// SIMATIC S7-200 project (STEP 7-Micro/WIN), CPU 224 AM REL 21.02

ORGANIZATION_BLOCK 主程序:OB1
TITLE=本MODBUS TCP 服务器库  可以建立两个 MODBUS TCP 服务器
// Socket：       填写1或者2通道（1=端口号502，2等于端口号503）
// MaxIO：        I 和Q 位最大数目（默认值128）
// MaxAI：        输入寄存器最大数目
// MaxHold：    保持寄存器最大数目
// ptrHold：       保持寄存器在V内存中的起始地址
// slaveAddr：  本服务端站号
// Error：           错误代码 =1 表示非法的数据地址 ， =2 表示错误的通信口 
// 
// 程序下载到PLC里面后需要重新上电
BEGIN
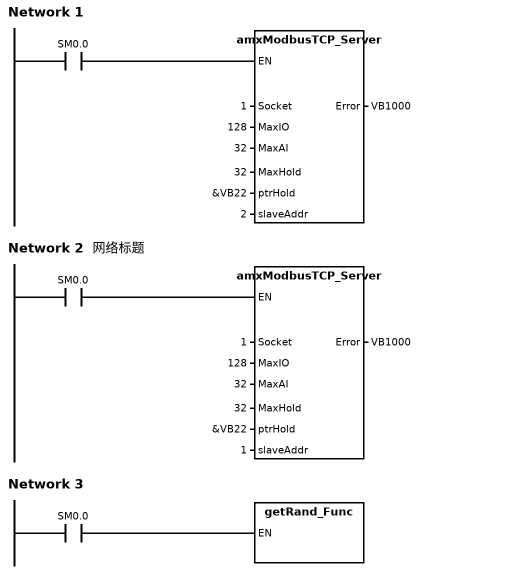
Network 1
LD     SM0.0
CALL   amxModbusTCP_Server:SBR1, 1, 128, 32, 32, &VB22, 2, VB1000
Network 2 // 网络标题
LD     SM0.0
CALL   amxModbusTCP_Server:SBR1, 1, 128, 32, 32, &VB22, 1, VB1000
Network 3
LD     SM0.0
CALL   getRand_Func:SBR0
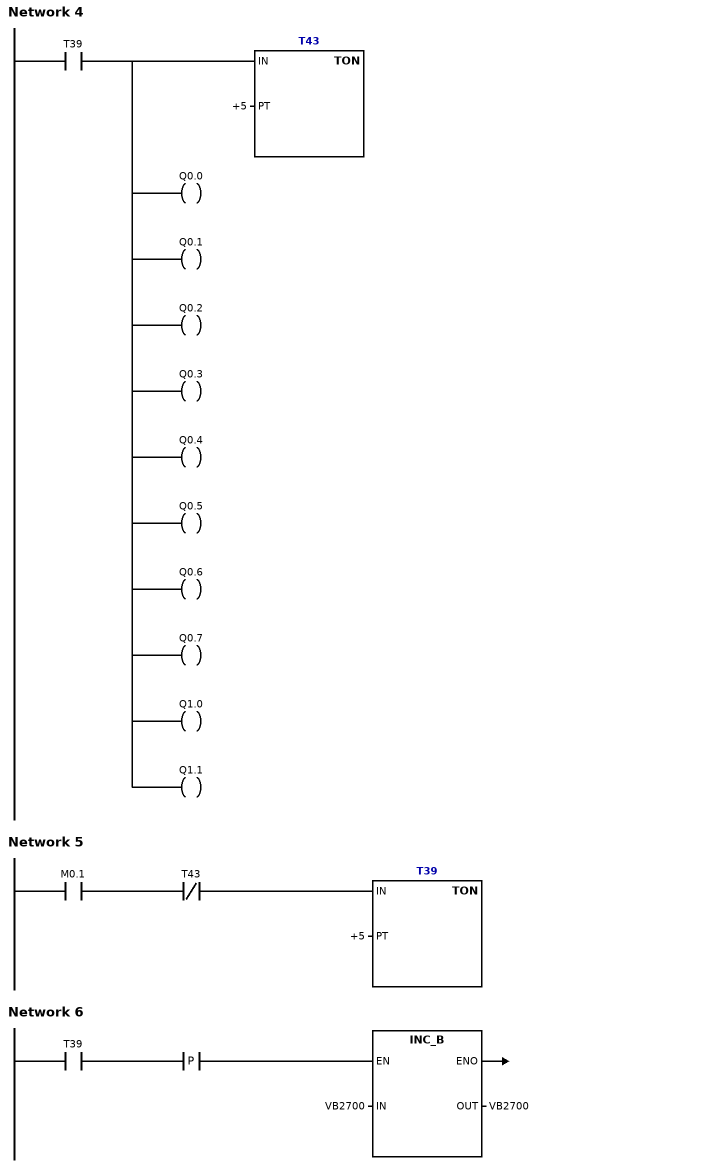
Network 4
LD     T39
TON    T43, +5
=      Q0.0
=      Q0.1
=      Q0.2
=      Q0.3
=      Q0.4
=      Q0.5
=      Q0.6
=      Q0.7
=      Q1.0
=      Q1.1
Network 5
LD     M0.1
AN     T43
TON    T39, +5
Network 6
LD     T39
EU
INCB   VB2700
END_ORGANIZATION_BLOCK

SUBROUTINE_BLOCK getRand_Func:SBR0
TITLE=
BEGIN
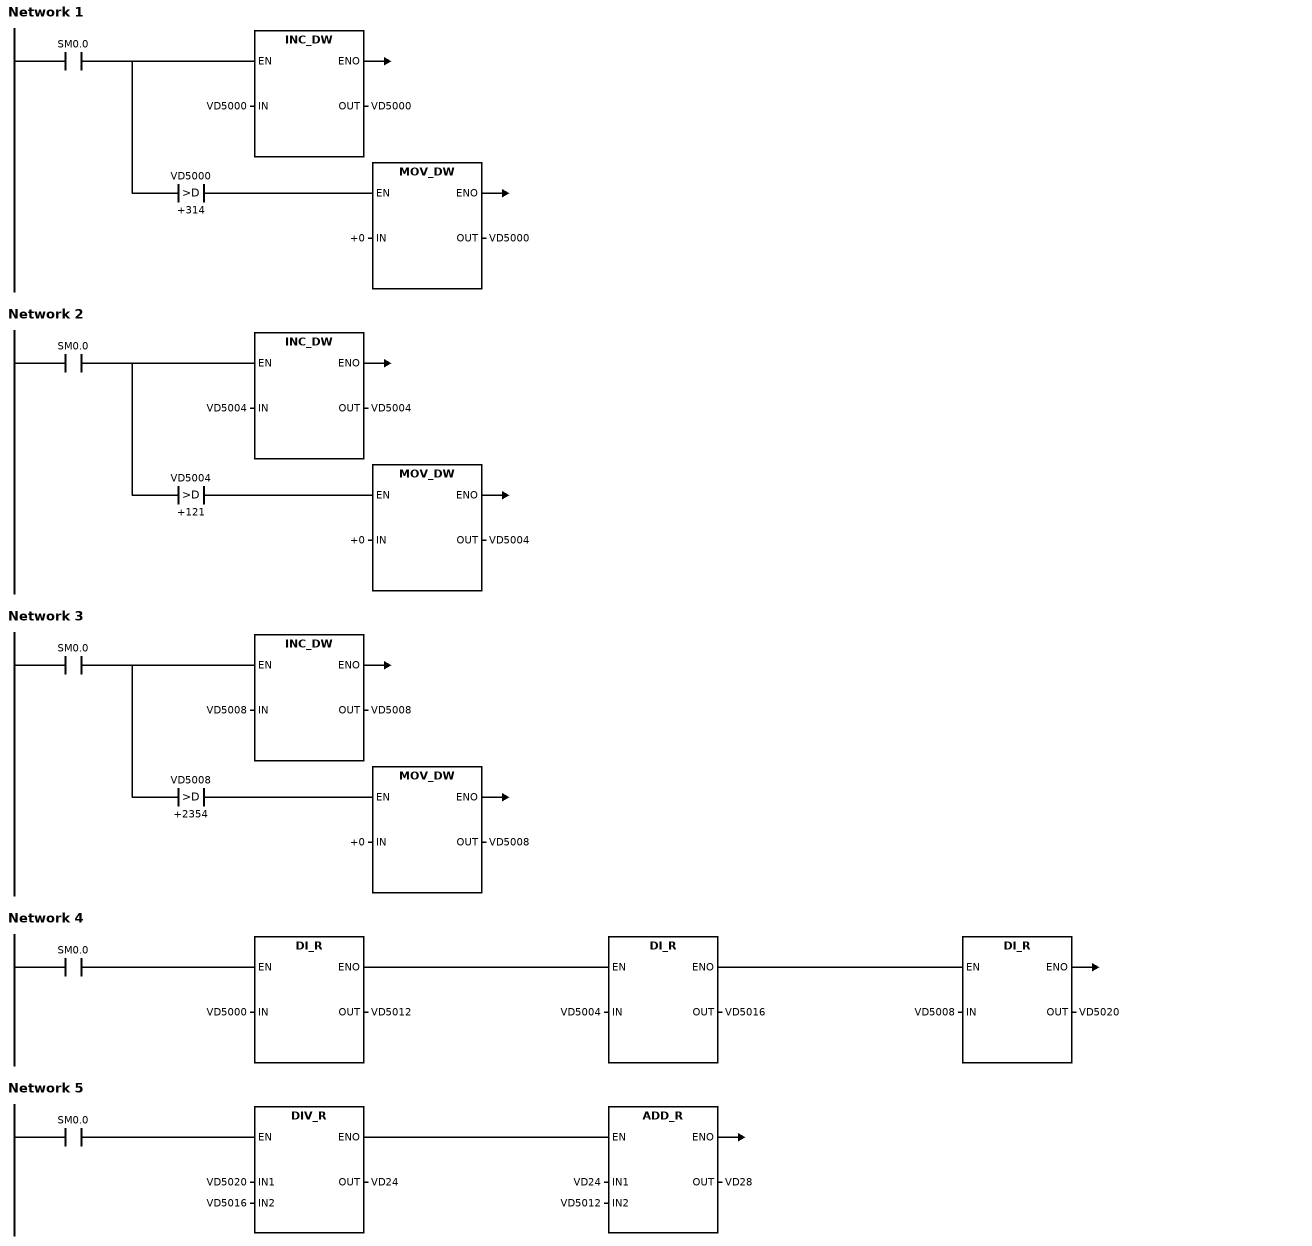
Network 1
LD     SM0.0
INCD   VD5000
AD>    VD5000, +314
MOVD   +0, VD5000
Network 2
LD     SM0.0
INCD   VD5004
AD>    VD5004, +121
MOVD   +0, VD5004
Network 3
LD     SM0.0
INCD   VD5008
AD>    VD5008, +2354
MOVD   +0, VD5008
Network 4
LD     SM0.0
DTR    VD5000, VD5012
AENO
DTR    VD5004, VD5016
AENO
DTR    VD5008, VD5020
Network 5
LD     SM0.0
MOVR   VD5020, VD24
AENO
/R     VD5016, VD24
AENO
MOVR   VD24, VD28
+R     VD5012, VD28
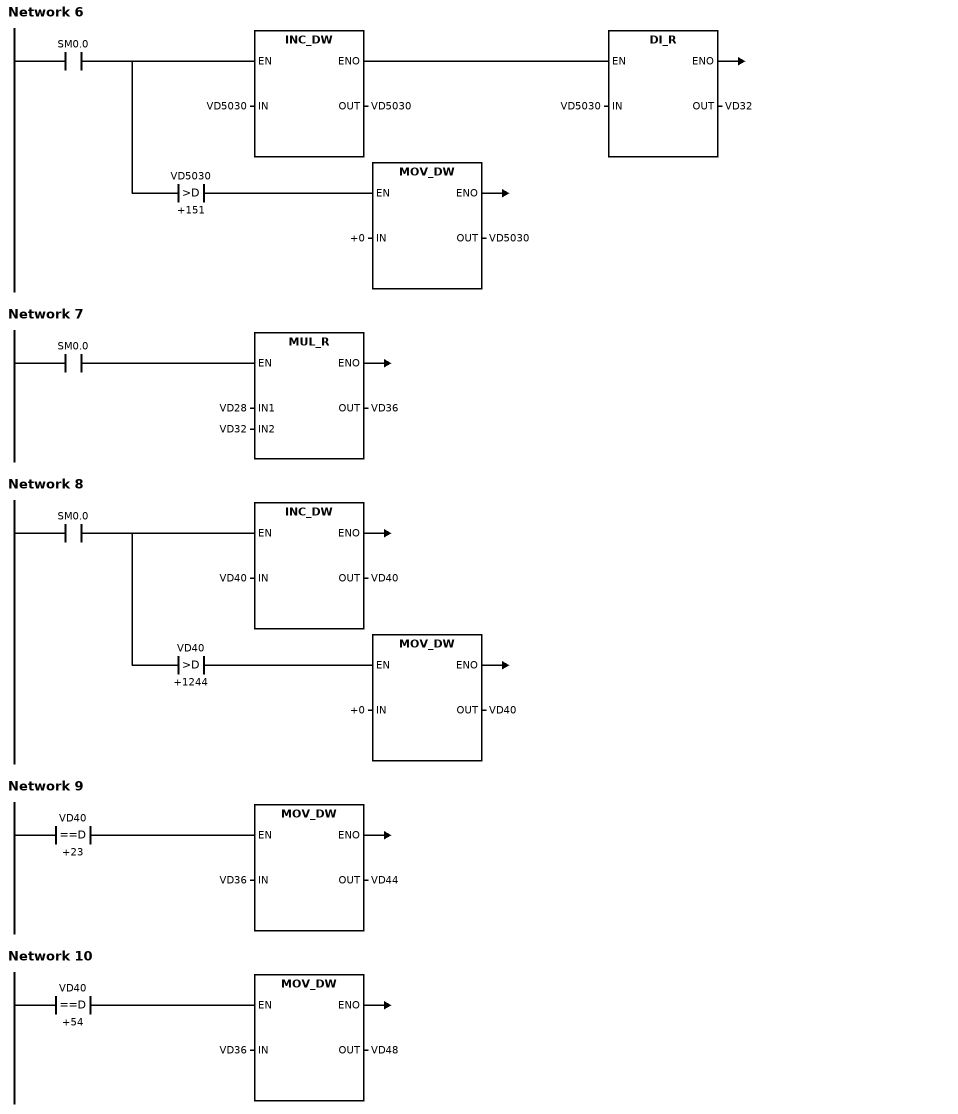
Network 6
LD     SM0.0
LPS
INCD   VD5030
AENO
DTR    VD5030, VD32
LPP
AD>    VD5030, +151
MOVD   +0, VD5030
Network 7
LD     SM0.0
MOVR   VD28, VD36
*R     VD32, VD36
Network 8
LD     SM0.0
INCD   VD40
AD>    VD40, +1244
MOVD   +0, VD40
Network 9
LDD=   VD40, +23
MOVD   VD36, VD44
Network 10
LDD=   VD40, +54
MOVD   VD36, VD48
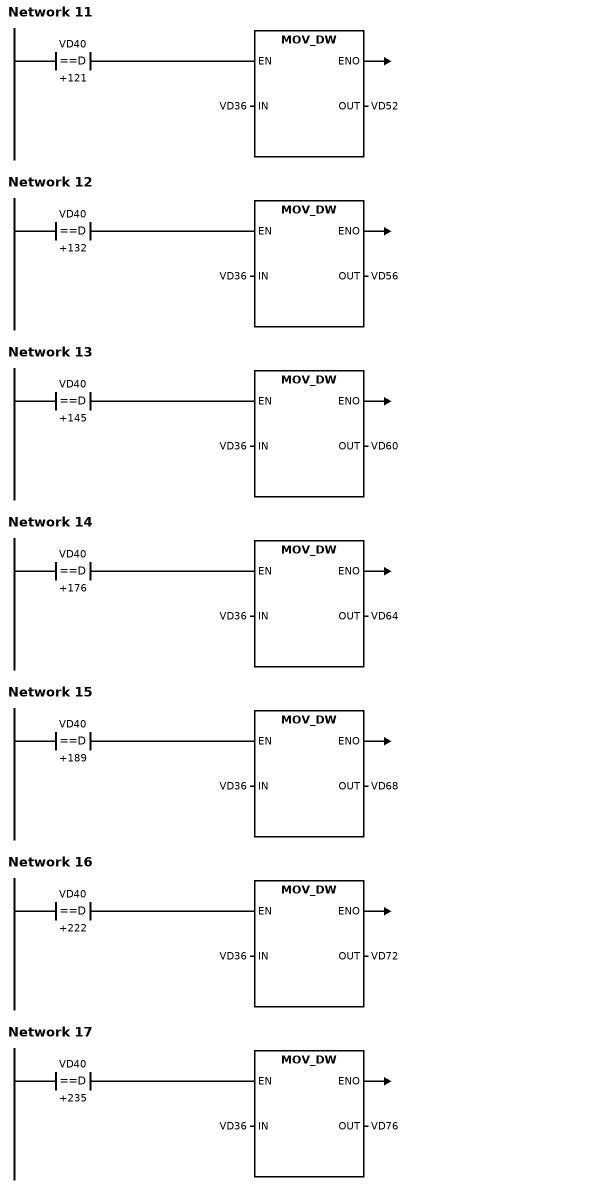
Network 11
LDD=   VD40, +121
MOVD   VD36, VD52
Network 12
LDD=   VD40, +132
MOVD   VD36, VD56
Network 13
LDD=   VD40, +145
MOVD   VD36, VD60
Network 14
LDD=   VD40, +176
MOVD   VD36, VD64
Network 15
LDD=   VD40, +189
MOVD   VD36, VD68
Network 16
LDD=   VD40, +222
MOVD   VD36, VD72
Network 17
LDD=   VD40, +235
MOVD   VD36, VD76
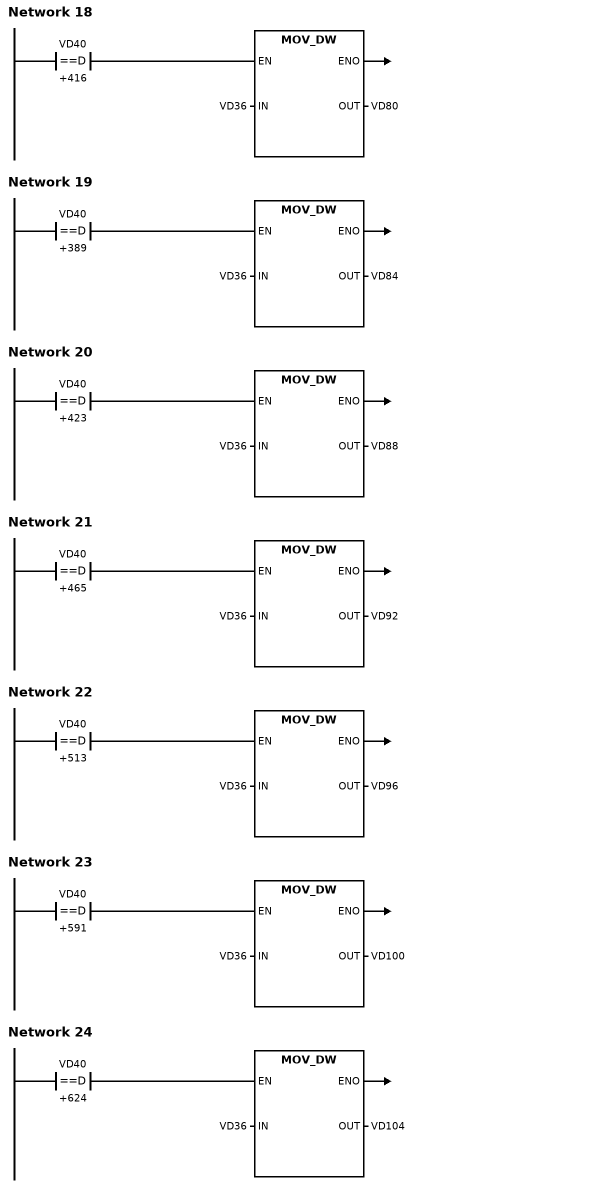
Network 18
LDD=   VD40, +416
MOVD   VD36, VD80
Network 19
LDD=   VD40, +389
MOVD   VD36, VD84
Network 20
LDD=   VD40, +423
MOVD   VD36, VD88
Network 21
LDD=   VD40, +465
MOVD   VD36, VD92
Network 22
LDD=   VD40, +513
MOVD   VD36, VD96
Network 23
LDD=   VD40, +591
MOVD   VD36, VD100
Network 24
LDD=   VD40, +624
MOVD   VD36, VD104
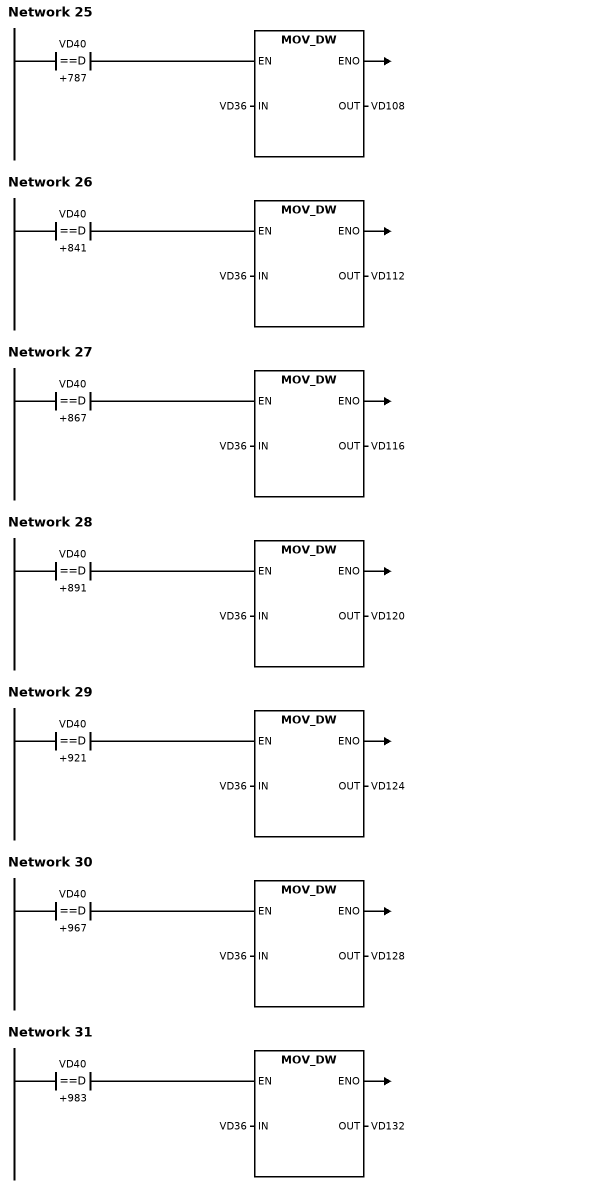
Network 25
LDD=   VD40, +787
MOVD   VD36, VD108
Network 26
LDD=   VD40, +841
MOVD   VD36, VD112
Network 27
LDD=   VD40, +867
MOVD   VD36, VD116
Network 28
LDD=   VD40, +891
MOVD   VD36, VD120
Network 29
LDD=   VD40, +921
MOVD   VD36, VD124
Network 30
LDD=   VD40, +967
MOVD   VD36, VD128
Network 31
LDD=   VD40, +983
MOVD   VD36, VD132
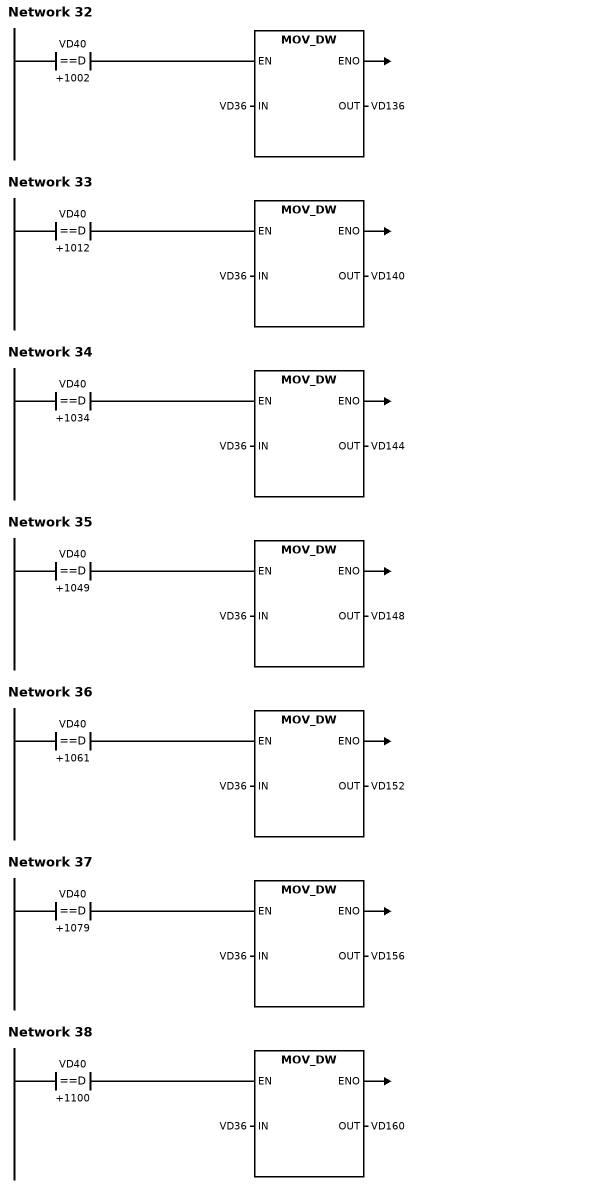
Network 32
LDD=   VD40, +1002
MOVD   VD36, VD136
Network 33
LDD=   VD40, +1012
MOVD   VD36, VD140
Network 34
LDD=   VD40, +1034
MOVD   VD36, VD144
Network 35
LDD=   VD40, +1049
MOVD   VD36, VD148
Network 36
LDD=   VD40, +1061
MOVD   VD36, VD152
Network 37
LDD=   VD40, +1079
MOVD   VD36, VD156
Network 38
LDD=   VD40, +1100
MOVD   VD36, VD160
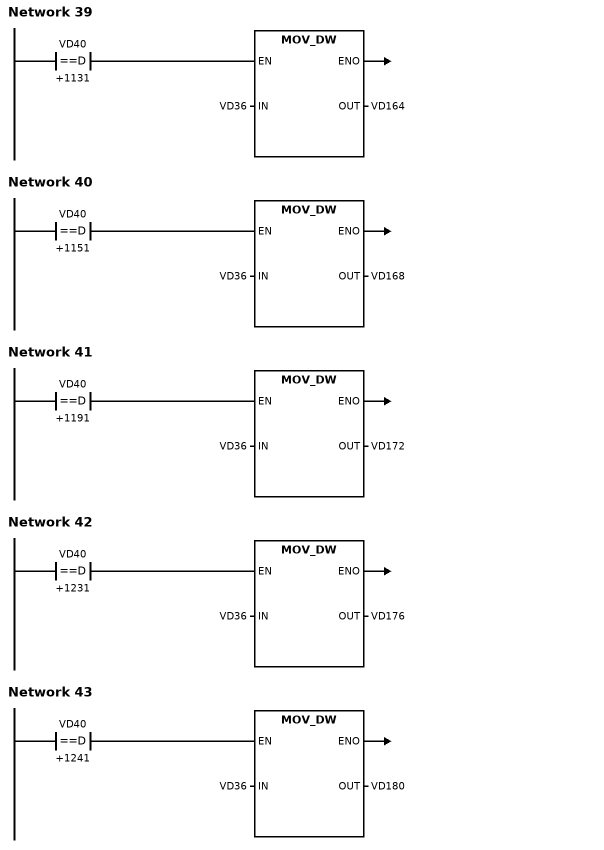
Network 39
LDD=   VD40, +1131
MOVD   VD36, VD164
Network 40
LDD=   VD40, +1151
MOVD   VD36, VD168
Network 41
LDD=   VD40, +1191
MOVD   VD36, VD172
Network 42
LDD=   VD40, +1231
MOVD   VD36, VD176
Network 43
LDD=   VD40, +1241
MOVD   VD36, VD180
Network 45 // Network Title
// Network Comment
END_SUBROUTINE_BLOCK

// SBR1: protected block, not included
